// TIA Portal V19 export
VAR_GLOBAL   // PLC tag table "TT - Clocks"
   Clock_Byte AT %MB255 : Byte;
   Clock_10Hz AT %M255.0 : Bool;
   Clock_5Hz AT %M255.1 : Bool;
   "Clock_2.5Hz" AT %M255.2 : Bool;
   Clock_2Hz AT %M255.3 : Bool;
   "Clock_1.25Hz" AT %M255.4 : Bool;
   Clock_1Hz AT %M255.5 : Bool;
   "Clock_0.625Hz" AT %M255.6 : Bool;
   "Clock_0.5Hz" AT %M255.7 : Bool;
END_VAR
